FUNCTION_BLOCK PIOC_Instantaneous_Overcurrent (* Composite Function Block Type *)
  (* Standard: 61499-2 *)
  (* Version 0.0, 12/10/2023, Cheyan, Schneider Electric, template *)
  PACKAGE Main;
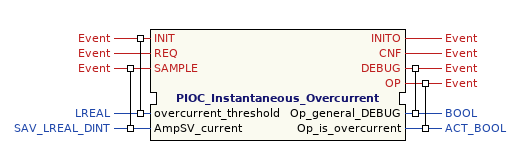
  EVENT_INPUT
    INIT WITH overcurrent_threshold; (* Initialization Request *)
    REQ; (* Normal Execution Request *)
    SAMPLE WITH AmpSV_current;
  END_EVENT
  EVENT_OUTPUT
    INITO; (* Initialization Confirm *)
    CNF; (* Execution Confirmation *)
    DEBUG WITH Op_general_DEBUG;
    OP WITH Op_is_overcurrent;
  END_EVENT
  VAR_INPUT
    overcurrent_threshold : LREAL;
    AmpSV_current : SAV_LREAL_DINT; (* Input event qualifier *)
  END_VAR
  VAR_OUTPUT
    Op_general_DEBUG : BOOL;
    Op_is_overcurrent : ACT_BOOL;
  END_VAR
  FBS
    FB1 : PIOC_Instantaneous_Overcurrent_Logic;
  END_FBS
  EVENT_CONNECTIONS
    INIT TO FB1.INIT;
    REQ TO FB1.REQ;
    FB1.INITO TO INITO;
    FB1.CNF TO CNF;
    FB1.DEBUG TO DEBUG;
    SAMPLE TO FB1.SAMPLE;
    FB1.OP TO OP;
  END_CONNECTIONS
  DATA_CONNECTIONS
    overcurrent_threshold TO FB1.overcurrentThreshold;
    FB1.debug_Op_general TO Op_general_DEBUG;
    AmpSV_current TO FB1.AmpSV;
    FB1.Op TO Op_is_overcurrent;
  END_CONNECTIONS
END_FUNCTION_BLOCK
